// TwinCAT 3 PLC project Untitled1
// ProgramVersion: 3.1.4024.0
// libraries:
//   Tc2_Standard, * (Beckhoff Automation GmbH)
//   Tc2_System, * (Beckhoff Automation GmbH)
//   Tc3_Module, * (Beckhoff Automation GmbH)
// project tree:
//   / PlcTask.TcTTO
//   POUs/ MAIN.TcPOU, Random.TcPOU
// real-time tasks:
//   TASK PlcTask: cycle T#10ms, priority 20, ADS port 350

CONFIGURATION Untitled1
    RESOURCE PLC ON TwinCAT3
        TASK PlcTask(INTERVAL := T#10ms, PRIORITY := 20);
        PROGRAM MAIN WITH PlcTask : MAIN;
    END_RESOURCE
END_CONFIGURATION

// ---- POUs/MAIN.TcPOU
PROGRAM MAIN
VAR
	sMessage : STRING;
	iTestIndex : INT;
	GenAleatoire : Random;
END_VAR;

// Premier test
CASE iTestIndex OF 
	1 : 
		sMessage := 'Bonjour jojo !';
	2 :
		sMessage := 'Au revoir';
	3 :
		sMessage :='';
END_CASE

// Second Test
GenAleatoire(iMinVal := 1, iMaxVal := 10, o_iResult => iTestIndex);

END_PROGRAM

// ---- POUs/Random.TcPOU
FUNCTION_BLOCK Random
VAR_INPUT
	iMinVal	: INT;
	iMaxVal	: INT;
END_VAR
VAR_OUTPUT
	o_iResult : INT;
END_VAR
VAR
	lrMidValue : LREAL;
	iMidValue : INT;
	drand		: drand;
END_VAR

drand(Seed := 0,Num => lrMidValue);

lrMidValue := lrMidValue * 10;
iMidValue := LREAL_TO_INT(lrMidValue);

IF iMidValue > iMinVal AND iMidValue < iMaxVal THEN
	o_iResult := iMidValue;
END_IF

END_FUNCTION_BLOCK
